// TIA Portal V20 export
DATA_BLOCK "F-DB_Axis"   // DB130, F_DB
// stored: AutoNumber false, InstanceOfName F-FB_Axis, InstanceOfType FB
"F-FB_Axis"
   // VAR
   //    LDrvSafe_SinaTlg903StatusAxis01_X : "LDrvSafe_SinaTlg903Status";
   //    LDrvSafe_SinaTlg903StatusAxis02_Y : "LDrvSafe_SinaTlg903Status";
   //    LDrvSafe_SinaTlg903StatusAxis03_ZM : "LDrvSafe_SinaTlg903Status";
   //    LDrvSafe_SinaTlg903StatusAxis04_B : "LDrvSafe_SinaTlg903Status";
   //    LDrvSafe_SinaTlg903StatusAxis05_U1 : "LDrvSafe_SinaTlg903Status";
   //    LDrvSafe_SinaTlg903StatusAxis06_U2 : "LDrvSafe_SinaTlg903Status";
   //    LDrvSafe_SinaTlg903StatusAxis07_V : "LDrvSafe_SinaTlg903Status";
   //    LDrvSafe_SinaTlg903StatusAxis08_W : "LDrvSafe_SinaTlg903Status";
   //    LDrvSafe_SinaTlg903StatusAxis09_ZL : "LDrvSafe_SinaTlg903Status";
   //    LDrvSafe_SinaTlg903ControlAxis01_X : "LDrvSafe_SinaTlg903Control";
   //    LDrvSafe_SinaTlg903ControlAxis02_Y : "LDrvSafe_SinaTlg903Control";
   //    LDrvSafe_SinaTlg903ControlAxis03_ZM : "LDrvSafe_SinaTlg903Control";
   //    LDrvSafe_SinaTlg903ControlAxis04_B : "LDrvSafe_SinaTlg903Control";
   //    LDrvSafe_SinaTlg903ControlAxis05_U1 : "LDrvSafe_SinaTlg903Control";
   //    LDrvSafe_SinaTlg903ControlAxis06_U2 : "LDrvSafe_SinaTlg903Control";
   //    LDrvSafe_SinaTlg903ControlAxis07_V : "LDrvSafe_SinaTlg903Control";
   //    LDrvSafe_SinaTlg903ControlAxis08_W : "LDrvSafe_SinaTlg903Control";
   //    LDrvSafe_SinaTlg903ControlAxis09_ZL : "LDrvSafe_SinaTlg903Control";
   // END_VAR
BEGIN
END_DATA_BLOCK
